(* CODESYS project lclsgeneral-v0.1.2.library
   Company: SLAC
   Version: 0.1.2
   Description: Generally useful POUs:
      - Logger
      - FB diagnostics
      - EtherCAT diagnostic
   Placeholder: LCLSGeneral
   Author: Alex Wallace
   Title: LCLS General

Project tree, tasks and I/O mapping:
  libraries: Tc2_EtherCAT, * (Beckhoff Automation GmbH); Tc2_Standard, * (Beckhoff Automation GmbH); Tc2_System, * (Beckhoff Automation GmbH); Tc2_TcpIp, * (Beckhoff Automation GmbH); Tc2_Utilities, * (Beckhoff Automation GmbH)
  Data types/
    Logger/
      data type E_MesgSevr
      data type E_MessengerState
      data type E_Subsystem
    Misc/
      data type ST_fbDiagnostics
      data type System_Struct
  POUs/
    Functions/
      function block FB_EcatDiag [ST]
      function block FB_Index [ST]: Dec, DecVal, Inc, IncVal
    Logger/
      function block FB_Logger [ST]: Manager, SocketSendTo
      function block FB_LogMessage [ST]
      function SYSTEM_TIME_TO_RFC3339 [ST]
  Version/
    global variables Global_Version
  global variables GVL_Logger
*)

// Data types/Logger/E_MesgSevr
TYPE E_MesgSevr :
(
	Emergency := 0, //system is unusable
	Alert	:= 1,	//action must be taken immediately
	Critical:= 2,	//critical conditions
	Error	:= 3,	//error conditions
	Warning	:= 4,	//warning conditions
	Notice	:= 5,	//normal but significant condition
	Info	:= 6,	//informational messages
	Debug	:= 7	//debug-level messages
) WORD;
END_TYPE

// Data types/Logger/E_MessengerState
TYPE E_MessengerState :
(
	Init := 0,
	CreateSocket	:= 1,
	Active	:= 2,
	CloseSocket := 3,
	Err	:= 10
);
END_TYPE

// Data types/Logger/E_Subsystem
TYPE E_Subsystem :
(
	NILVALUE := 0,
	VACUUM := 1,
	MPS := 2,
	MOTION := 3,
	FIELDBUS := 4,
	SDS := 5
)WORD;
END_TYPE

// Data types/Misc/ST_fbDiagnostics
TYPE ST_fbDiagnostics :
STRUCT
	asResults	:	ARRAY [1..20] OF STRING;
	resultIdx	:	FB_Index := (
		LowerLimit := 1,
		UpperLimit := 20
	);
	fString	:	FB_FormatString;
END_STRUCT
END_TYPE

// Data types/Misc/System_Struct
TYPE System_Struct :
STRUCT

	xswAlmRst 		: BOOL;(* Global Alarm Reset - EPICS Command *)
	xAtVacuum 	    : BOOL;(* System At Vacuum *)
	xFirstScan	    : BOOL; (* Bit set for one scan only during startup. Used for initialization. *)
	xOverrideMode	: BOOL; //This bit is set when using the override features of the system
	xIOState        : BOOL; (* ECat Bus Health *)

END_STRUCT
END_TYPE

// Version/Global_Version
{attribute 'TcGenerated'}
// This function has been automatically generated from the project information.
VAR_GLOBAL CONSTANT
	{attribute 'const_non_replaced'}
	{attribute 'linkalways'}
	stLibVersion_LCLS_General : ST_LibVersion := (iMajor := 0, iMinor := 1, iBuild := 2, iRevision := 0, sVersion := '0.1.2');
END_VAR

// GVL_Logger
VAR_GLOBAL
	g_psLogHost	: T_IPv4Addr := '172.21.32.9';
	g_udpSyslog	:	UDINT := 514;
	gMesgBuffer	:	ARRAY [0..cMesgArraySize] OF T_MaxString; //maybe this should be persistent...
	gsCurrentTime	:	T_MaxString := cNILVALUE;
	gsHostName	:	T_MaxString := cNILVALUE;
	fbLogMessage : FB_LogMessage;
	gfbBuffer 			:	FB_StringRingBuffer;
END_VAR
VAR_GLOBAL CONSTANT
	acsSubsystems	:	ARRAY [0..5] OF STRING := 
	['-', 'VACUUM', 'MPS', 'MOTION', 'FIELDBUS', 'SDS'];
	cNILVALUE	:	STRING(1) := '-';
	cMesgArraySize : INT := 50;
	cwFacility: WORD := 20; // local4
	// Syslog Version
	cwSyslogVer: WORD := 1;
END_VAR

// POUs/Functions/FB_EcatDiag
FUNCTION_BLOCK FB_EcatDiag
VAR_INPUT
	///Connect this to an AMSNETID structure as a PLC input. Then link the input to the AMSNETID name in the master info.
	i_AMSNetId: AMSNETID; 
	i_xFirstPass: BOOL;
END_VAR
VAR_OUTPUT
	q_xAllStatesGood: BOOL;
END_VAR
VAR
	sNetId: T_AmsNetId;
	astTermStates: ARRAY[1..256] OF ST_EcSlaveState;
	fbGetAllSlaveStates: FB_EcGetAllSlaveStates;
	ftReset: F_TRIG;
	iterator: INT;
END_VAR

(* 
Ecat bus diagnostic tool
2015-11-4 Alex Wallace
This function block checks the states of all slaves on the ecat bus network, 
it could be modified to export the states of the slaves on an individual basis,
but for now it sets the output boolean true if all slaves are OP and false otherwise.
To start the block provide a falling edge on the first pass boolean input.
*)

//Create the net ID string
sNetID := F_CreateAmsNetId(i_AMSNetId);

//Query the state of all terminals, collect in astTermStates
ftReset(CLK:=fbGetAllSlaveStates.bBusy OR i_xFirstPass);
fbGetAllSlaveStates.bExecute := ftReset.Q;
fbGetAllSlaveStates(sNetId:=sNetId, pStateBuf := ADR(astTermStates), cbBufLen:=SIZEOF(astTermStates));
//Keep checking...

//Cycle through each entry in the array and check if we have anyone not in OP and that the link state is good.
// If so, then set our global IO bad boolean.
IF fbGetAllSlaveStates.nSlaves > 0 THEN
	q_xAllStatesGood := TRUE;
FOR iterator := 1 TO (UINT_TO_INT(fbGetAllSlaveStates.nSlaves) -1) BY 1
	DO
	IF NOT( (astTermStates[iterator].deviceState = EC_DEVICE_STATE_OP) AND (astTermStates[iterator].linkState = EC_LINK_STATE_OK)) THEN
		q_xAllStatesGood := FALSE;
	END_IF
END_FOR
END_IF

END_FUNCTION_BLOCK

// POUs/Functions/FB_Index
FUNCTION_BLOCK FB_Index
VAR_INPUT
	LowerLimit : INT := 1;
	ValInc : INT := 1;
	UpperLimit	:	INT := 1;
END_VAR
VAR_OUTPUT
	
END_VAR
VAR
	Val	:	INT := LowerLimit;
END_VAR

(* Index FB
A. Wallace 2016-9-3

Why doesn't beckhoff have this as a builtin type?
*)

;

ACTION Dec:
Val := Val - ValInc;
IF Val < LowerLimit THEN Val := UpperLimit; END_IF
END_ACTION

METHOD DecVal : INT
VAR_INPUT
END_VAR
Dec();
DecVal := Val;
END_METHOD

ACTION Inc:
// Dont use this, use ValInc
Val := Val + ValInc;
IF Val >  UpperLimit THEN Val := LowerLimit; END_IF
END_ACTION

METHOD PUBLIC IncVal : INT
VAR_INPUT
END_VAR
Inc();
IncVal := Val;
END_METHOD

END_FUNCTION_BLOCK

// POUs/Logger/FB_Logger
FUNCTION_BLOCK FB_Logger
VAR_INPUT
	i_CloseSocket	:	BOOL := FALSE;
	i_bReset		:	BOOL := FALSE;
END_VAR
VAR
	fbUDPSocketManager	:	FB_ConnectionlessSocket;
	udpSocket			:	T_HSOCKET;
	fbUDPSocketSend		:	FB_SocketUdpSendTo;
	sOutgoingMesg		:	T_MaxString;
	eState				:	E_MessengerState;
	stDiag				:	ST_fbDiagnostics;
	rtReset				:	R_TRIG;
	fbGetSystemTime		:	FB_LocalSystemTime := (bEnable := TRUE);
	fbGetHostName		:	FB_GetHostName := (bExecute := TRUE, sNetID := '');
	ctuSentSomething	:	CTU := (PV := 100);
	rtSocketSendErr		:	R_TRIG;
END_VAR
VAR CONSTANT

END_VAR

(* Syslog Logger
A. Wallace 2016-9-3

This is used to pass PLC notification messeges to a syslog server.

This POU constantly attempts to send out messages from the global buffer.
*)

gfbBuffer.pBuffer := ADR(gMesgBuffer); 
gfbBuffer.cbBuffer:= SIZEOF(gMesgBuffer);

fbGetSystemTime(); 
IF fbGetSystemTime.bValid THEN
	gsCurrentTime := SYSTEM_TIME_TO_RFC3339(fbGetSystemTime.systemTime);
ELSE
	gsCurrentTime := cNILVALUE;
END_IF

fbGetHostName();
IF NOT (fbGetHostName.bBusy OR fbGetHostName.bError) THEN
	gsHostName := fbGetHostName.sHostName;
ELSE
	gsHostName := cNILVALUE;
END_IF

IF i_CloseSocket THEN 
	eState := CloseSocket; 
END_IF

rtReset(CLK:=i_bReset);
IF rtReset.Q THEN
	eState := CreateSocket;
	i_bReset R= i_bReset;
END_IF

rtSocketSendErr(CLK:=fbUDPSocketSend.bError);

CASE eState OF
	Init:
		;
	CreateSocket:
		fbUDPSocketManager.nLocalPort := g_udpSyslog;
		fbUDPSocketManager.bEnable := TRUE;
		
		IF fbUDPSocketManager.eState = eSOCKET_CREATED THEN
			eState := Active;
		ELSIF fbUDPSocketManager.bError THEN
			eState := Err;
			fbUDPSocketManager.bEnable := FALSE;
			stDiag.fString( sOut=>stDiag.asResults[stDiag.resultIdx.IncVal()], sFormat:='Socketmanger error in createsocket: %d', arg1:=F_UDINT(fbUDPSocketManager.nErrID));
		//ELSE
			//eState := Err;
			//stDiag.fString( sOut=>stDiag.asResults[stDiag.resultIdx.IncVal()], sFormat:='Something else happened in createsocket -> error');
		END_IF
	Active:
		IF fbUDPSocketManager.eState = eSOCKET_TRANSIENT  OR 
			fbUDPSocketManager.bError THEN
			eState := Err; 
			stDiag.fString( sOut=>stDiag.asResults[stDiag.resultIdx.IncVal()], sFormat:='Socketmanager error in active: %d', arg1:=F_UDINT(fbUDPSocketManager.nErrId));
		END_IF
		
		// While the socket is active, go ahead and send whatever is in the buffer
		IF rtSocketSendErr.Q THEN
			eState := Err;
			stDiag.fString( sOut=>stDiag.asResults[stDiag.resultIdx.IncVal()], sFormat:='Socket send error: %d', arg1:=F_UDINT(fbUDPSocketSend.nErrId));
		ELSIF gfbBuffer.nCount > 0 AND NOT fbUDPSocketSend.bBusy THEN
			gfbBuffer.A_RemoveHead(getValue=>sOutgoingMesg);
			fbUDPSocketSend.bExecute := TRUE; //reset in the action after busy goes true
			IF sOutgoingMesg <> '' THEN
				ctuSentSomething(CU:=TRUE);
			END_IF
		ELSIF gfbBuffer.nCount = 0 OR fbUDPSocketSend.bBusy THEN
			stDiag.fString( sOut=>stDiag.asResults[stDiag.resultIdx.IncVal()], sFormat:='Waiting to send');
			ctuSentSomething(CU:=FALSE);
		ELSE
			eState := Err;
			stDiag.fString( sOut=>stDiag.asResults[stDiag.resultIdx.IncVal()], sFormat:='Something else happened in active -> error');
		END_IF
		
	CloseSocket:
		fbUDPSocketManager.bEnable R= i_CloseSocket;
		IF fbUDPSocketManager.eState = eSOCKET_CLOSED THEN
			eState := Init;
		ELSIF fbUDPSocketManager.bBusy AND NOT fbUDPSocketManager.bEnable THEN
			;
		ELSIF fbUDPSocketManager.bError THEN
			eState := Err;
		ELSE
			eState := Err;
		END_IF
	Err:
		eState := Init;
		stDiag.asResults[stDiag.resultIdx.IncVal()] := 'Moving back to Init state from Error';
END_CASE



Manager();
SocketSendTo();

ACTION Manager:
fbUDPSocketManager(hSocket => udpSocket);
END_ACTION

ACTION SocketSendTo:
fbUDPSocketSend.hSocket := udpSocket;
fbUDPSocketSend.sRemoteHost := g_psLogHost;
fbUDPSocketSend.nRemotePort := g_udpSyslog;
fbUDPSocketSend.pSrc := ADR(sOutgoingMesg);
fbUDPSocketSend.cbLen := SIZEOF(sOutgoingMesg);
fbUDPSocketSend();
fbUDPSocketSend.bExecute R= fbUDPSocketSend.bBusy;
END_ACTION

END_FUNCTION_BLOCK

// POUs/Logger/SYSTEM_TIME_TO_RFC3339
FUNCTION SYSTEM_TIME_TO_RFC3339 : STRING
VAR_INPUT
	tCurrentTime	:	TIMESTRUCT;
END_VAR
VAR
END_VAR

SYSTEM_TIME_TO_RFC3339 := CONCAT(REPLACE(SYSTEMTIME_TO_STRING(tCurrentTime), 'T', 1, 11), 'Z');

END_FUNCTION

// POUs/Logger/FB_LogMessage
FUNCTION_BLOCK FB_LogMessage
VAR_INPUT	
	i_sMsg	:	STRING;
	i_eSevr	:	E_MesgSevr;
	i_eSubsystem	:	E_Subsystem; //In-lieu of App-name in the RFC-5424
END_VAR
VAR
	i_sPID	:	STRING := cNILVALUE;	//Not currently used
	i_sMSGID	:	STRING := cNILVALUE; //Not currently used
	i_sSD	:	STRING := cNILVALUE; //Not currently used
	fbFormatString		:	FB_FormatString;
	sPRIVAL				: 	T_MaxString := cNILVALUE;
	sPID				: 	T_MaxString := cNILVALUE;
	sSubsystem			: 	T_MaxString := cNILVALUE;
	wSyslogVer			: 	WORD := cwSyslogVer;
	sSD					: 	T_MaxString := cNILVALUE;
	sMsg				: 	T_MaxString := cNILVALUE;
END_VAR

gfbBuffer.putValue := '';
gfbBuffer.pBuffer := ADR(gMesgBuffer);
gfbBuffer.cbBuffer := SIZEOF(gMesgBuffer);

fbFormatString.sFormat := '<%s> %d %s %s %s %s BOM%s';

sPRIVAL := LEFT( WORD_TO_STRING(cwFacility * 8 + i_eSevr), 5);
sPID := cNILVALUE;
sSubsystem := acsSubsystems[i_eSubsystem];
wSyslogVer := cwSyslogVer;
sSD := i_sSD;
sMsg := i_sMsg;
//bad language ahead, sorry
fbFormatString.arg1 := F_STRING(sPRIVAL);
fbFormatString.arg2 := F_WORD(wSyslogVer);
fbFormatString.arg3 := F_STRING(gsCurrentTime);
fbFormatString.arg4 := F_STRING(sSubsystem);
fbFormatString.arg5 := F_STRING(sPID);
fbFormatString.arg6 := F_STRING(sSD);
fbFormatString.arg7 := F_STRING(sMsg);
fbFormatString( sOut=>gfbBuffer.putValue);
gfbBuffer.A_AddTail();

END_FUNCTION_BLOCK
